(* PLC project PLC, Beckhoff Automation GmbH TwinCAT PLC Control 3.5.21.60 *)
(* stored: creationDateTime 2026-08-05T00:25:24.016427, modificationDateTime 2026-08-05T00:25:24.016427 *)

FUNCTION_BLOCK FB_InitTCPIP
VAR_INPUT
END_VAR
VAR_OUTPUT
END_VAR
VAR
	sSrvNetID 		: T_AmsNetID := '';(* TwinCAT TCP/IP server network address *)
	fbCloseAll		: FB_SocketCloseAll;
END_VAR

            (* On PLC reset or program download close all created/opened sockets/connections *)
fbCloseAll( sSrvNetID := sSrvNetID, bExecute:= bInitTCPIP );
IF fbCloseAll.bBusy OR fbCloseAll.bError THEN
	RETURN;
END_IF
bInitTCPIP := FALSE;
          
END_FUNCTION_BLOCK
